PROGRAM DeleteLastInstruction
VAR
END_VAR

IF GVL_MOTION.EXT_CTR.CMDDEL THEN
	GVL_MOTION.EXT_CTR.CMDDEL					:= FALSE;
	//QueueEnd contains no data
	IF GVL_MOTION.ScriptEnd <> 0 THEN
		GVL_MOTION.ScriptEnd 					:= GVL_MOTION.ScriptEnd - 1;
		GVL_MOTION.Script[GVL_MOTION.ScriptEnd]	:= GVL_MOTION.EmptyInstruction;
		GVL_MOTION.EXT_CTR.CMDDEL 				:= FALSE;
	ELSE
		//error msg
		GVL_MOTION.EXT_CTR.CMDDEL 				:= FALSE;
	END_IF

END_IF

END_PROGRAM

(* stored: Version 1.1.0.1, ProductVersion 3.1.4026.18
   POU DeleteLastInstruction: Id {98abe00f-97f9-49d5-a61d-9227ab1e0d6f}, SpecialFunc None *)
